(* IEC 61131-3 sources: ml2plc/benchmarks/st (part 21) *)

(* ---- ResNet2_straton.st ---- *)
FUNCTION_BLOCK ResNet2_FB

    (* Model Inputs/Outputs *)
VAR_INPUT
    input_data : REAL;
END_VAR

VAR_OUTPUT
    output_data : ARRAY[0..2] OF REAL;
END_VAR

VAR
    CONSTANT weights_0 : ARRAY[0..31] OF REAL := [0.446109116, -0.253379464, -0.341707826, 0.579259038, -0.196502939, 0.384631842, 0.528063476, -0.174200714, 0.4646855, 0.173207715, 0.330620855, -0.331686378, -0.31313917, -0.175854653, 0.48702389, 0.211235866, -0.0733348131, -0.239896551, 0.256497949, 0.395332277, -0.227466539, 0.452796817, -0.260912657, 0.231070071, -0.198892906, -0.148901105, 0.498160481, 0.427462339, 0.327300549, 0.239787996, -0.318450183, 0.391796708];
    CONSTANT bias_0 : ARRAY[0..31] OF REAL := [0.0780105293, 0, 0, -0.0437059142, 0, -0.0844902843, -0.0905284137, 0, -0.0596597679, 0.15236482, 0.109405488, 0, 0, 0, 0.0613273531, 0.0716272369, 0, 0, -0.0532285497, -0.055359453, 0, -0.0825184509, 0, -0.0527263731, 0, 0, -0.108202934, -0.0454206392, -0.0738661438, -0.0547046475, 0, -0.0875417367];
    CONSTANT weights_1 : ARRAY[0..1023] OF REAL := [-0.0672997385, 0.123918496, 0.0261855032, -0.207488403, 0.295382023, -0.205328912, -0.220387012, 0.309004188, -0.151001543, 0.397226214, 0.266850084, -0.0449176431, -0.0748620778, -0.0714222938, 0.0556719527, -0.21978052, -0.141455054, 0.0768866539, 0.148485273, 0.179841518, -0.120705262, 0.242057636, -0.0162528157, 0.0534217693, 0.107853472, 0.139660329, -0.0586810037, -0.0446375608, -0.244673312, 0.135248959, -0.0232865997, 0.291286677, 0.133107841, -0.0169415176, 0.072581023, -0.0316966772, -0.246254802, 0.156484276, 0.230665118, -0.022424221, 0.0690721869, 0.0099068284, 0.280228585, 0.282496542, 0.0474284887, -0.0939033031, -0.157858804, -0.0393083394, -0.200870991, 0.196391314, -0.0571665317, 0.0700698793, 0.0415192544, 0.283202559, 0.108373076, 0.18269524, -0.117297322, -0.287417442, -0.045781225, -0.200513572, -0.0697987527, 0.0264480114, 0.169026285, -0.0959516168, -0.0716886669, 0.297260195, -0.136756331, -0.189135864, -0.0970409364, -0.303627491, -0.0101010799, -0.273864031, -0.111413628, -0.124916166, 0.199581772, -0.264739096, 0.0937647521, -0.0471192598, 0.0671662092, -0.184105843, 0.2014893, -0.205362201, 0.273994476, -0.00908637047, -0.0441014767, -0.200558037, -0.0472564399, -0.0810055733, -0.137171343, -0.175276652, -0.303469598, 0.0569872558, -0.122404516, 0.132641941, -0.117922872, -0.0366746485, -0.271390259, -0.181193858, 0.154695168, 0.123995334, 0.300765067, -0.0419366695, 0.30564639, 0.0560056716, -0.13017562, 0.371984065, 0.0800307393, -0.243357852, 0.242418826, 0.2982063, 0.390265286, -0.29279983, 0.229600817, -0.105995312, 0.147868991, -0.282524794, 0.0784076452, 0.33515355, -0.0324381292, -0.127563611, -0.0404234231, 0.117910236, -0.268573463, 0.437732875, 0.205221027, -0.0789395124, 0.142241478, 0.318100512, -0.00765234232, 0.155244231, 0.229942471, 0.139751703, 0.167155415, -0.224905014, -0.253680557, 0.111216456, 0.166616023, 0.195199996, 0.26445052, -0.0218468606, 0.165077895, -0.305733055, 0.161665052, -0.280608475, 0.0925857723, -0.0801890641, 0.0903935134, -0.0246531367, 0.207986385, 0.244579464, -0.218942255, 0.254853576, -0.184336007, -0.259816915, 0.0658665895, 0.0739070773, 0.0859895349, 0.2244443, 0.303090066, -0.168849394, -0.117300168, -0.203983143, -0.516042411, -0.240961015, 0.320624799, 0.22011438, 0.155475706, 0.167489037, -0.223099396, 0.514761925, -0.0340227485, -0.135615855, 0.2276887, 0.100083739, -0.046878662, 0.00446370244, -0.16629912, 0.0464164019, -0.124795854, -0.211745948, -0.339682132, 0.560887516, -0.0539340675, -0.495146632, -0.154791906, 0.391963482, 0.0478856824, 0.300241709, -0.00436666375, -0.272856534, 0.473389745, 0.0918120444, -0.186532736, 0.169220388, -0.33542341, -0.13656354, 0.184764907, 0.121988617, -0.0807672292, 0.17290619, -0.0137443729, 0.403550833, -0.169839054, -0.199931324, 0.0710707009, 0.208184093, 0.194795758, 0.102081329, -0.135433197, -0.0341715217, -0.174149469, -0.269304931, -0.428490847, 0.436180294, -0.21050106, 0.136596486, 0.203933746, 0.305774748, 0.0526449233, 0.366092116, 0.38880232, -0.124543056, 0.399355233, -0.0542085133, -0.0242547095, 0.259555787, 0.169075102, -0.0785467029, -0.257587254, 0.0482283533, -0.303375334, 0.262526006, 0.195120007, 0.159601986, 0.0649527013, 0.289143413, 0.0153873265, -0.289190114, 0.184705019, 0.0448786616, -0.0187006891, 0.129755288, -0.000189214945, -0.12248905, -0.238008529, -5.98728657e-05, -0.159052655, -0.128630728, -0.127178386, -0.0828053951, 0.117196888, 0.291492611, 0.125405937, 0.0925316215, 0.24035868, 0.189899445, 0.0789665282, -0.114477828, 0.101446815, 0.0898142457, -0.0724863037, 0.267957658, -0.0225918293, -0.103431433, -0.176787034, 0.33514151, -0.276106536, -0.216690555, -0.0109675825, -0.237743527, 0.345496029, 0.0550661683, -0.281188637, -0.281930357, 0.0209647622, 0.173377007, -0.275085509, 0.442110121, -0.27953425, -0.269451231, -0.159710318, -0.0268889349, 0.261009961, 0.292426825, 0.00604014285, -0.039501071, 0.44544968, 0.385405064, -0.103716165, 0.197616503, 0.140080914, -0.190431833, -0.142311439, 0.338202953, -0.302250057, 0.00575613463, 0.237771541, 0.321618259, -0.248187274, 0.254863501, -0.0786112323, -0.256906897, 0.165188715, 0.00759845972, 0.196345091, 0.0205950439, 0.0259478632, 0.278409153, 0.269123256, -0.0704165474, -0.102515385, 0.143988624, -0.253235906, 0.00062259991, 0.0771465674, 0.102807239, -0.180491194, -0.0101891756, 0.108349077, 0.0780294985, -0.128736287, -0.236025348, -0.0358681642, -0.00330647826, -0.0861312822, 0.181077912, 0.117443472, 0.356189668, 0.188092053, 0.0508594029, -0.273949802, -0.00910276547, -0.274905294, -0.250903606, 0.241061077, 0.215696722, -0.0816203058, -0.21879968, 0.408205211, -0.246976987, -0.136179954, 0.320423037, 0.119813651, 0.349625587, -0.225764737, 0.353475153, -0.0903084055, -0.0600670241, -0.0816910192, -0.246967867, -0.125283241, 0.104817316, 0.194935232, -0.22541666, 0.139627814, -0.162285402, -0.139945656, -0.273778468, 0.154627442, -0.0709560364, -0.0483515859, 0.139850885, 0.26585874, 0.170851052, 0.0655213594, 0.275238186, 0.110014439, 0.241464347, 0.139358073, 0.225116462, 0.0450653136, 0.0663165748, 0.0984885991, -0.161821276, -0.253443301, -0.0401959717, -0.0450824797, -0.0893658102, -0.191750675, -0.114205316, -0.113555402, -0.032099843, -0.251139253, 0.0875837803, -0.0385817885, 0.14630121, -0.126950979, 0.15461868, 0.0945681036, 0.257601351, -0.131864205, -0.28712675, 0.231681079, 0.230294853, 0.261832148, 0.193466842, -0.301149845, -0.201477766, -0.236950368, 0.146894932, 0.042988807, -0.112412274, -0.255944818, 0.210005194, -0.0656734258, -0.126614377, 0.040821135, -0.045797646, -0.244730994, 0.25871709, -0.10164924, 0.0108816624, -0.263333112, -0.15512611, -0.265041053, -0.0407094359, 0.288093776, 0.244367093, 0.108738452, 0.0884629488, 0.125704706, 0.0346384346, 0.0489260256, -0.117135048, -0.0452102125, 0.123711288, 0.0750169158, 0.03458938, 0.0375772119, -0.160466671, 0.153726101, 0.299916059, 0.205223113, 0.099450469, 0.168587625, -0.170589864, 0.0105227232, -0.00761330128, -0.192904949, -0.0217333436, -0.0766484588, -0.236247391, 0.273411483, -0.171270818, 0.0562030673, 0.0808565915, -0.302630812, -0.171502382, -0.250153184, -0.201328039, 0.0215679221, -0.11872448, 0.342555076, -0.0201337449, -0.260737449, 0.308816582, 0.0652882904, 0.391782105, -0.11709775, -0.221956342, -0.125762343, -0.19962348, 0.0793167502, -0.301425576, -0.173867315, -0.0441781282, 0.120754406, 0.144720495, 0.0815581903, -0.196122408, -0.0626295954, -0.113548383, 0.175504923, 0.145190552, 0.0946770385, 0.151647747, 0.217094958, -0.203452721, -0.038656652, 0.101846643, -0.10814628, 0.108325951, 0.0775899515, -0.195024371, -0.241803467, -0.0457298718, 0.133528113, 0.42471084, -0.146245062, 0.120418303, -0.263231128, -0.14939186, -0.00569485081, -0.211991802, -0.110631473, -0.122159302, 0.211433142, -0.0213046074, 0.239424616, -0.172884226, 0.302616417, -0.0958690196, -0.198209673, 0.235887215, 0.201637536, 0.257626355, -0.261320055, -0.050790146, 0.1605165, -0.277989268, 0.27792275, 0.015366096, -0.21359621, -0.169574067, 0.255636603, -0.159326404, -0.242564619, -0.0658581853, 0.23809275, -0.0649103522, 0.0572633445, -0.233979613, -0.0433489978, 0.209428161, 0.100888282, 0.0781544745, 0.227146178, -0.216204301, 0.0940120816, -0.0834899247, -0.0717138499, 0.10444814, 0.0668695271, -0.227245539, -0.0815511048, -0.0642618835, 0.160572588, -0.186493456, -0.0400582254, 0.170362264, 0.274944872, -0.138044864, -0.0465166271, -0.0316170156, 0.141667455, -0.0781259239, 0.222043961, -0.292664409, -0.09773013, -0.267205209, -0.013055563, -0.268664062, -0.258037746, -0.233674765, -0.197328925, -0.181961954, 0.210466653, -0.074807182, 0.0213672519, 0.135242075, 0.29159227, 0.0965499282, -0.208291113, 0.170358896, -0.271036923, -0.0950112939, 0.118789613, -0.160189778, 0.0534884632, 0.165033877, -0.235269174, 0.0221406221, -0.0631530881, 0.175863415, -0.224407643, 0.23844102, -0.225643396, -0.149267823, 0.046709083, -0.22471258, 0.342396617, 0.382626325, 0.086022675, -0.111780778, 0.0649216473, 0.117322743, -0.22994262, -0.162323654, -0.309645176, 0.0411821902, 0.0823624283, 0.25201419, -0.16624178, 0.0215016305, -0.05505725, -0.279398203, -0.231971473, 0.473751515, -0.0695412159, 0.169299603, -0.216064066, 0.215218201, -0.102295764, 0.0126560032, 0.330998242, -0.238440096, -0.0759054124, 0.235605121, 0.0308294296, -0.205652803, -0.153373122, 0.21992442, -0.107053734, 0.449966788, -0.246368393, 0.303302258, -0.164613053, 0.281154096, 0.251495153, -0.0526953936, 0.128691703, -0.0415357351, -0.123309121, -0.125063479, -0.243296653, -0.200463638, 0.263173014, 0.0401532613, -0.0997288153, -0.00675202301, 0.272087842, -0.0488012917, -0.241687015, 0.2161116, 0.181204066, 0.383062124, -0.152072236, -0.175835103, 0.382474452, -0.0213172268, 0.0795238912, 0.293702573, 0.117500931, 0.302794188, -0.048030436, -0.0943690389, 0.280748278, 0.106655836, 0.27533105, -0.0209568441, 0.091119647, -0.0680115521, -0.0532403588, 0.00992289186, -0.135216832, 0.184090495, -0.198157549, 0.246385604, -0.183580667, 0.212307185, 0.134317905, -0.0904083997, -0.208351851, -0.00371128321, 0.016589433, 0.232418746, 0.173685908, -0.290628523, 0.275564283, -0.165179148, 0.177294314, 0.159701705, -0.0396937132, 0.0288962126, 0.0287567955, -0.0214288533, 0.406184524, 0.188659236, -0.137733087, 0.288018227, -0.376283169, 0.211254671, 0.0125238299, -0.182050586, -0.136293024, 0.244678944, 0.0101755811, -0.0860448629, -0.192576677, 0.144176096, 0.246334776, -0.0542725213, -0.319506258, 0.249152645, 0.300927252, -0.216155916, -0.263445467, 0.501632154, -0.0983170569, 0.490621924, 0.377952546, 0.182914823, 0.517102718, 0.292947888, 0.176778853, -0.0453032255, -0.292213202, 0.116734773, 0.0421213508, 0.0886447132, 0.164180636, 0.177889407, -0.0874125361, -0.28499952, -0.253518581, -0.0666396618, -0.191444427, 0.00308844447, -0.124373332, 0.0720646083, -0.201085448, 0.0728932619, -0.0851670355, 0.268443495, 0.291759223, -0.296979994, 0.15201956, 0.18446368, 0.128499776, 0.301611513, 0.200069577, 0.305754751, 0.23328355, 0.0512740016, 0.211027056, -0.0285782218, 0.28756842, -0.235887274, -0.201257139, -0.0654639155, -0.0219288748, 0.517582595, 0.142651647, -0.0918668807, -0.480128437, 0.445097446, -0.039173007, 0.206185371, -0.291620851, 0.289303392, -0.0353964828, -0.0932732373, 0.243763298, -0.168045878, 0.301816911, -0.454546899, -0.350679219, 0.389303118, -0.154629558, 0.0356258824, 0.217119068, 0.375954688, -0.216656104, 0.0966599658, 0.472218037, 0.24505803, 0.474726588, 0.287663907, -0.00348621607, 0.0777794719, 0.248905092, 0.304142505, 0.069024086, -0.00871711969, -0.17508626, 0.138942629, 0.0450723171, 0.222106844, 0.166393012, -0.285030186, -0.146981001, -0.173450544, 0.169468075, 0.101617634, 0.14248687, -0.211429179, -0.281644136, -0.21104835, 0.0707558692, -0.161577746, -0.179358691, -0.292363435, -0.0184406638, -0.0107237101, -0.0946408212, 0.119637281, 0.232440859, -0.188967675, -0.288388342, -0.0585837662, -0.0083989203, -0.189461887, 0.260625094, 0.0797997415, -0.0345056653, -0.273636639, -0.295552671, 0.111130029, 0.2143493, 0.0990378559, 0.0820131898, 0.219696254, -0.176936746, 0.194112211, -0.185160339, 0.20026961, 0.299959809, 0.132246137, -0.226150692, -0.165659562, 0.0304536223, 0.0551926792, -0.18758285, -0.00389325619, 0.120256096, -0.0793661326, 0.182034016, -0.0968718678, 0.210053414, 0.0536976159, -0.058866784, 0.032423377, -0.245521799, -0.0334720314, -0.476026595, 0.0220496655, 0.0105779376, 0.360177249, 0.226633102, 0.0757015273, -0.438258886, 0.176172927, 0.234365493, -0.22066617, -0.0561640561, -0.19579117, 0.355135053, -0.0497905016, 0.265808195, 0.0921390355, -0.219965175, -0.145613924, -0.043286223, 0.386870444, 0.10977602, -0.286260992, -0.0710007846, 0.302653104, 0.0277191214, 0.354971856, 0.129811853, 0.066929847, 0.00035183024, 0.216759875, -0.00531771779, 0.0594547167, -0.344661593, 0.29841271, 0.25737071, 0.322826356, -0.0608721077, 0.436551511, 0.163451761, -0.0346164703, 0.0586311519, 0.15674755, -0.115996219, -0.274861425, 0.0137932487, -0.306024313, -0.0696883276, -0.209392697, 0.0805150419, 0.0509290658, -0.110743746, 0.117124185, -0.110970736, 0.0164447147, -0.281959713, 0.179450154, 0.0630740449, -0.140035346, 0.324055582, -0.0899775475, 0.239219546, 0.400147587, -0.245016277, -0.0488338172, -0.457950622, -0.0780736506, 0.17666854, 0.395307273, 0.230418056, 0.454527378, -0.443111569, 0.103358082, 0.297938734, -0.270894229, 0.082223542, -0.0515313447, 0.152576774, 0.115509778, 0.130205333, -0.00376668572, 0.107549623, 0.0414021388, -0.118665934, 0.193046421, -0.00821468234, -0.455872506, -0.0179270804, 0.283343107, 0.0154615017, 0.157088995, 0.450618804, 0.226627737, 0.52094692, 0.0691082925, 0.00625914335, -0.190991536, -0.192506939, -0.114632443, 0.270887166, 0.426719934, -0.0118926466, 0.026724346, -0.384286642, -0.0412942842, -0.111217633, 0.153527528, 0.222803086, -0.186998546, -0.0981789753, 0.031683743, -0.136033341, 0.196271867, -0.295513868, -0.422320575, -0.319054574, 0.253908068, -0.0470398366, -0.359538227, -0.262141675, 0.556122601, -0.0490951799, 0.422659874, 0.243652195, 0.0135763288, 0.204732895, 0.504005373, 0.0145732462, -0.151889265, 0.295809776, 0.0527801514, -0.29109928, -0.0319833457, 0.00571236014, -0.108667865, -0.243677378, -0.187169373, -0.033985436, 0.0185488462, 0.0218675137, 0.078579098, 0.148238659, 0.0607049465, -0.0328954756, 0.164118737, 0.103054196, 0.0620963275, 0.228370219, -0.245889515, 0.00231522322, 0.00149768591, 0.207119197, -0.0681625307, -0.263822019, -0.0741106719, 0.303110272, 0.0252650976, 0.0528681874, 0.288920611, -0.0862795711, -0.183671564, -0.415967107, 0.0277608335, -0.0389414392, 0.509281099, -0.0653216392, 0.08415059, -0.146404579, 0.027331626, 0.0637321174, 0.0652593672, 0.119661465, 0.0570983589, 0.490790248, 0.0708687305, 0.0192686319, -0.135138795, 0.0672079623, -0.0580277219, -0.241328657, 0.495732963, 0.038197875, -0.444418669, -0.260325283, 0.0363532118, -0.0319354162, 0.21500051, 0.259890407, -0.136209637, 0.280829757, 0.164074123];
    CONSTANT bias_1 : ARRAY[0..31] OF REAL := [0, -0.00853045937, 0.126876727, 0, -0.0861710161, -0.0860414207, 0, 0.0468492433, 0.136715055, 0.0599241219, 0, -0.0130215548, -0.0051236595, 0, 0.0153312925, 0, -0.0135006029, 0, 0.184726223, 0.136625856, 0.102708332, -0.0912417546, 0, 0.150348634, 0, -0.0932127312, -0.00915876683, -0.0861517116, -0.0181769449, 0, -0.0608111285, -0.0683147013];
    CONSTANT weights_2 : ARRAY[0..1023] OF REAL := [-0.204679489, -0.135256469, 0.28196618, -0.0638390034, -0.174786299, 0.126281202, -0.209497452, 0.222915739, -0.0468465388, -0.216639012, -0.250750899, -0.280927479, -0.259657174, 0.0156140029, -0.235811859, 0.278314084, 0.0742395222, 0.290134758, -0.258248925, 0.0707915723, -0.302265584, -0.0793548822, 0.109813094, -0.20324108, 0.223869294, -0.052572906, 0.205616981, 0.102512896, -0.0969290286, 0.140410602, 0.241890162, 0.0239737928, -0.291626126, -0.216462642, 0.157533735, 0.21785447, -0.1888697, 0.0757077038, 0.222794265, -0.106055737, -0.192728728, -0.188463166, -0.182898849, -0.0930845514, -0.0597978532, 0.0867448747, -0.0387444645, -0.290577084, 0.0780397058, 0.0745291114, -0.172289535, 0.0823122859, -0.134248555, 0.252856761, -0.205714047, -0.102416694, -0.178794965, 0.0999448672, -0.00859764218, 0.243844897, 0.236200243, -0.113696873, -0.201874301, -0.113263831, -0.0378434174, -0.227657393, 0.0797862336, 0.333367527, -0.299939692, -0.0166706592, -0.125392675, 0.253749698, -0.355483234, 0.426590443, 0.558343112, 0.409482211, 0.187631369, 0.227338403, 0.285558254, 0.252233982, -0.349539638, -0.098085463, -0.0745894611, -0.260414094, 0.113806494, -0.36481443, -0.241131589, 0.0945619047, 0.452752471, 0.101931356, -0.30287379, 0.0321633108, 0.130271345, -0.0806449354, -0.210663259, -0.220049694, -0.17137076, -0.191594154, 0.301324457, -0.2250586, -0.253617704, 0.232058376, 0.077934593, 0.180609912, -0.139309749, -0.0280079544, 0.253463835, 0.244393975, 0.237231284, -0.20984596, 0.212327093, 0.264635891, 0.180089056, 0.218266934, 0.212391943, 0.280880839, 0.180849433, 0.106197894, 0.147727877, 0.018728435, 0.257006079, -0.206631452, -0.212920159, 0.166844428, -0.246302903, -0.00446945429, 0.247142047, -0.00678348541, -0.236221522, 0.277348638, 0.0965815783, -0.226228476, -0.0891875252, 0.40643695, 0.465085387, -0.152245566, 0.196031243, 0.140979126, -0.171359077, -0.0893353596, 0.454827428, 0.261000603, -0.299895495, -0.23500298, 0.0234229378, -0.060218025, 0.203745693, 0.122152202, -0.211209461, 0.0520563908, 0.10854879, 0.0593966246, -0.275008678, 0.0641941652, 0.481133044, -0.256873101, -0.285603046, 0.479949445, -0.135300189, 0.478868186, -0.406574875, 0.403340727, 0.0558100753, 0.225551426, 0.41712141, 0.00127660832, -0.0283386484, 0.0520305708, 0.500523508, -0.206790835, -0.362006932, -0.000284219335, 0.11284703, 0.130605608, -0.264846265, 0.133523747, 0.398929954, -0.00425994396, 0.44960174, 0.376377463, 0.2425109, 0.241941929, 0.246711314, 0.170248806, -0.264131367, 0.369570494, 0.443199039, 0.12817663, -0.182199731, 0.224466771, 0.257635802, 0.184784427, -0.0534651875, 0.114040047, -0.26297009, -0.137307927, 0.191011965, -0.224709436, 0.193394721, 0.134513915, 0.179350376, -0.188209772, 0.0368874371, -0.000262796879, -0.189553499, 0.11833626, 0.199825972, -0.168204218, 0.146432757, 0.232580811, 0.149660856, 0.122925818, 0.217384726, -0.143141761, 0.278794497, -0.0659557879, 0.2359505, 0.0733537376, -0.181416214, -0.24697648, 0.156488746, 0.163566709, 0.154782563, 0.16413027, -0.0641885176, 0.162349254, -0.165244937, -0.00756666251, -0.0619688965, 0.125170499, -0.164782301, 0.0368066728, 0.438915193, 0.369288772, -0.17342855, 0.372006238, 0.180813387, -0.0500442386, 0.181848824, 0.35768488, 0.33091262, 0.201537341, 0.0606543608, 0.183581203, -0.329741299, 0.19205898, -0.124992542, -0.203194737, 0.0749375671, 0.129340827, 0.0689797103, 0.0523179248, -0.232102171, 0.106971428, -0.164516747, -0.028096538, 0.26692003, -0.416765064, 0.146759704, 0.123076126, -0.313440531, -0.270631313, -0.449947, -0.0287845936, -0.411788732, 0.478075385, 0.478816599, 0.373561949, 0.0675536245, -0.204258502, 0.171388388, 0.416653246, -0.222486272, 0.212794915, -0.0879907608, -0.0584020466, 0.141890928, 0.153230354, -0.432367802, 0.197440714, 0.350558281, 0.383365989, -0.0781740323, 0.186996579, -0.195837736, -0.393867284, -0.12553376, 0.146623254, 0.07671763, 0.391239494, 0.192586288, 0.0520732291, 0.0479876958, -0.180293262, 0.0687054694, -0.309032947, -0.118887261, 0.162971631, 0.232025594, -0.115431778, 0.0105950609, -0.149042457, 0.275376558, 0.276807368, 0.161677882, -0.246772081, -0.0466549844, -0.0590618029, -0.0781350955, 0.0737073869, 0.299358219, -0.288225114, 0.166770518, 0.396302283, 0.349194467, -0.121977806, -0.203997999, 0.382262409, -0.154711246, 0.298326313, 0.0719448328, -0.0823758692, -0.230296239, 0.0475671887, 0.0851532519, 0.0975213349, 0.238155454, 0.174278498, -0.175005093, -0.265223473, -0.263997346, -0.198879018, 0.0115664899, 0.0591326654, -0.149858981, -0.109177634, -0.178252071, -0.00203052163, 0.268845469, 0.0775773823, 0.0275386274, -0.206349224, -0.136653408, -0.15385583, -0.155029312, -0.282329679, -0.222141564, 0.0748182833, 0.255190402, 0.171676189, 0.146660447, -0.149523973, -0.0342544094, 0.0865873992, 0.196472615, 0.0615327805, -0.201127067, -0.0292131901, 0.0689860284, 0.217757076, 0.220056325, 0.0298993532, -0.246281326, 0.0094137406, -0.205014378, 0.133170396, -0.00583136268, 0.230486065, -0.18984434, -0.265659779, 0.177857876, 0.21923694, 0.050457865, 0.178938717, 0.267668396, 0.179177284, 0.168444872, -0.172058687, -0.269957036, 0.198731601, 0.0808540285, -0.210361779, -0.203446448, -0.0371791422, -0.115300179, -0.0115000643, -0.15966849, -0.0855638981, -0.0802038908, 0.0730054528, 0.182234421, 0.0919757187, -0.0438024141, -0.284938186, -0.161267102, 0.0511448085, 0.201944143, 0.151732385, 0.11750789, 0.0223256852, 0.208975583, -0.0789252073, -0.249366164, 0.0771737546, -0.210034892, 0.0630125329, 0.282773703, -0.168602288, -0.228485093, -0.197542459, 0.227408201, 0.00968745165, 0.114427835, 0.251161247, -0.189475894, 0.0572520047, -0.0855299979, -0.012209028, 0.255862862, 0.0658447444, 0.279396147, 0.229320735, -0.0213460028, 0.0183748901, 0.0143043697, 0.175676167, 0.00535911322, -0.227714136, 0.210220248, -0.193221331, -0.244543672, -0.148611754, -0.190139264, 0.197188467, 0.112814814, 0.271459013, -0.28341198, 0.283254832, 0.194213003, 0.270252079, 0.0488406122, -0.137301132, 0.214347333, 0.213200539, -0.180703938, -0.128120601, -0.206830531, 0.0404673219, -0.0389949307, 0.0506746434, -0.0645795316, 0.0863745436, -0.00896019023, -0.200361013, -0.0323581994, 0.0325997397, -0.0739912689, 0.17362231, 0.0897462815, -0.12044479, 0.31924805, -0.27516371, 0.31264019, -0.11941921, 0.353853881, -0.0860883221, 0.218072325, -0.0713869631, 0.0661892593, 0.123493522, 0.154916063, -0.141882941, 0.142999113, 0.401889205, 0.386382669, 0.239116251, -0.228276312, 0.0787872225, -0.29939267, 0.00509946654, -0.115147322, -0.259926319, -0.0525318086, 0.0664702356, 0.0423623323, 0.1990951, 0.0846948028, 0.30295524, 0.181253284, -0.0447692871, -0.0963983834, -0.239262372, -0.053407073, 0.271961659, 0.0432170928, 0.129507035, -0.0613849461, -0.161630079, 0.223844141, -0.168244153, 0.131808519, -0.132705614, -0.0131464303, -0.0498532057, 0.0134880841, 0.205623835, 0.0286743045, -0.304037899, 0.297517449, 0.0676321685, 0.0823118389, -0.130943239, -0.0981799364, 0.0825493038, 0.092310302, 0.132190675, -0.0180039704, 0.222785085, 0.137986481, 0.289361268, 0.0720570758, 0.129101664, -0.140128732, -0.168845177, -0.126143813, -0.0213747621, 0.038553644, -0.303022981, 0.163347989, -0.20824483, -0.0491371453, 0.0485385358, -0.253569454, 0.0288275182, -0.0582758486, 0.0342372358, 0.00962677598, 0.231157124, -0.240408048, -0.21099937, -0.0426646173, 0.294546098, -0.245215863, -0.18224594, -0.0182284415, 0.135243684, 0.0727446079, 0.217568904, 0.166266769, 0.138461411, -0.2175951, 0.129577965, -0.230868846, -0.152226597, -0.131347224, 0.0510773361, 0.00408044457, 0.169953823, -0.0437824726, 0.163264632, -0.270352781, 0.212604791, -0.205052525, -0.202281937, -0.173584491, 0.248010248, 0.00338539481, 0.141827911, -0.117097601, 0.289717048, -0.261541098, 0.175698817, 0.103879333, -0.116942108, 0.125927597, -0.27946943, 0.133731633, 0.0409375429, 0.11390619, -0.0837004408, 0.199883446, 0.202443495, 0.146647006, 0.265037954, 0.18095395, 0.323377252, 0.111219957, 0.210307673, 0.0840765238, 0.301873416, 0.252628654, 0.176735342, -0.225448921, -0.00881180167, 0.264034539, -0.0576801077, -0.207668871, -0.0362603888, 0.183284, -0.222751856, 0.029674856, 0.253859907, -0.301360816, 0.276103348, 0.159531534, 0.09506578, 0.296914607, -0.0876111984, -0.218210489, -0.224868655, -0.276840299, 0.170778424, -0.0902170613, 0.026544407, 0.0524329469, 0.139356345, 0.337209821, 0.343271613, 0.106872618, 0.247088611, -0.146878138, -0.140349343, 0.319549531, 0.265812397, -0.0614267886, 0.176764369, -0.295758694, 0.00160560687, 0.142407343, -0.17890656, 0.00188067136, -0.179448411, 0.323931873, 0.14950569, 0.112876579, -0.0789793506, -0.254204988, -0.249873608, -0.111487955, 0.233570397, -0.0383268632, -0.220227048, 0.188659593, 0.138276428, -0.391264945, -0.219422072, 0.119032457, -0.324904621, -0.149002716, 0.260387927, 0.512180686, 0.343798786, 0.246067539, -0.213445902, 0.343288749, -0.0358869024, -0.0598138869, 0.0849777758, -0.229632109, 0.0804907382, -0.207954884, -0.246657565, -0.152553603, 0.230183572, 0.258402884, 0.605133116, -0.000907221751, 0.40813598, 0.138139337, -0.394745469, -0.245143875, -0.356614888, -0.278564036, 0.51167649, -0.167552158, 0.0385506786, 0.30153054, 0.178012431, 0.491966486, -0.226964116, 0.249466941, -0.31189698, -0.212363005, 0.12730749, 0.107616968, 0.245273083, -0.0632424355, -0.107013598, 0.400151312, -0.126116946, 0.443775713, 0.0567636304, -0.0484892353, 0.225377142, 0.17650643, -0.16261822, -0.350496858, 0.21365118, 0.0242102928, -0.272912949, 0.144263998, 0.183707282, 0.235746235, 0.106295653, -0.0331136882, 0.117457211, -0.0399730206, 0.0439910293, 0.0704419613, -0.169385076, 0.137371719, 0.183431178, 0.0584154129, -0.266066253, 0.0112705529, -0.0212856233, 0.223700017, -0.0228022039, 0.0189183056, -0.0324111879, -0.155158073, -0.22306934, 0.11734134, 0.288133234, 0.275658756, -0.179903343, 0.296819836, -0.187510654, -0.154961348, 0.275978237, 0.267136604, 0.1356273, 0.0229957998, -0.166162252, -0.0112787187, 0.271157116, 0.504267514, -0.0745441094, -0.128601953, 0.396112651, -0.0514549389, -0.0184277389, -0.0510308333, -0.151744619, 0.0578206517, 0.451091677, 0.449969262, 0.439691722, -0.121170506, -0.107776523, 0.201376095, 0.392380595, -0.37306577, -0.182681888, -0.082582891, -0.0752992257, -0.0241405126, 0.154176563, 0.0456010364, -0.200354218, 0.186367407, 0.0181775708, -0.202771991, 0.154682621, -0.182058185, -0.219726712, 0.059972316, -0.343565434, 0.209741443, -0.222851798, -0.199444413, -0.02868554, 0.235248834, -0.304307938, 0.161286384, 0.201732069, -0.0422318876, -0.157119676, -0.224580228, 0.067997545, -0.125626177, 0.0241714716, -0.0759897828, -0.0502993762, -0.296199769, 0.243887156, -0.267505169, 0.138399065, -0.233483225, 0.246404737, -0.174308226, -0.137947485, 0.101638436, 0.124087334, -0.114575863, 0.096797049, 0.0372642577, 0.0244682431, -0.10504967, 0.0597021282, -0.243710384, 0.346117526, -0.191104233, 0.00756108714, 0.360030293, 0.254576176, 0.380814731, -0.170184657, 0.0216305014, 0.169229582, -0.0979294181, -0.174209282, 0.345129073, 0.113265961, -0.108804695, 0.363609046, 0.212997556, -0.033747524, -0.068172805, 0.198910668, 0.258692235, 0.252833068, 0.2392544, -0.0721322894, -0.333581597, 0.0375342928, -0.110548787, 0.326079488, 0.0975811481, 0.314479381, 0.147384316, 0.424212158, 0.162820056, 0.279910028, -0.149647564, -0.113421351, 0.122204378, 0.0914485157, -0.11268647, 0.0712843239, -0.0754816532, -0.113101743, 0.129354239, -0.0762300938, -0.294329286, 0.018773675, 0.0962105021, -0.0627630502, -0.139184624, -0.0883929282, 0.192166761, -0.0048656296, 0.0775612146, 0.014094159, -0.227728426, 0.16301775, 0.248803243, 0.139576599, -0.236111104, -0.134085178, -0.0108638359, 0.0713160485, 0.000784546137, 0.0634449497, -0.285768718, 0.540881157, -0.0152861401, 0.196317405, 0.0716606081, -0.118341036, 0.377459377, 0.0323503166, 0.503604591, -0.325088292, -0.351278603, -0.345217735, 0.345662981, -0.115596712, -0.213419259, -0.0567794181, 0.110530913, -0.281917006, 0.269924909, 0.134860232, -0.183613077, 0.222686723, 0.22196804, 0.130703807, -0.137397841, 0.095159784, 0.382972747, -0.257635623, -0.114726156, 0.219153389, -0.274423659, 0.193779275, -0.378756016, 0.55745393, -0.273371994, 0.153506696, 0.347348154, -0.0390162319, -0.0190924518, 0.0466835201, 0.338260919, -0.289644122, -0.045777481, -0.0979495496, -0.109888777, -0.159528181, -0.315120131, 0.0249667857, 0.3593283, -0.266355038, 0.329570562, 0.0659172311, 0.141647443, 0.172656283, 0.413104653, -0.0921770632, -0.309635311, 0.0745841414, -0.0158826876, 0.159715265, 0.280772299, 0.185895413, -0.224144131, 0.0355212055, -0.0401628911, 0.258820683, 0.020608902, -0.00089943409, -0.126454577, -0.187050238, 0.0248265862, 0.21769926, -0.039658457, -0.193980694, 0.191328883, 0.251601726, 0.238136321, 0.247954696, -0.122940779, 0.133804053, 0.12044853, -0.00639125705, 0.084846288, -0.250858724, 0.184372365, -0.0337354839, 0.173017561, 0.185794771, -0.136319786, -0.154326752, 0.161565125, -0.0733977556, -0.261118054, 0.237281889, -0.284483045, 0.259607047, -0.118910857, 0.319470137, -0.0940027982, 0.167246327, 0.15437226, 0.423810035, 0.453898102, 0.2123539, 0.515671432, -0.263677806, -0.384399831, -0.276800603, 0.440641314, -0.115233019, 0.273297697, -0.149060681, 0.187632188, -0.0750807822, 0.393690765, -0.15505597, -0.0574740916, 0.110269904, 0.451854825, 0.121877313, -0.311037689, 0.205216989, -0.07337486, 0.234148517, -0.108864084, 0.344401598, -0.256927043, 0.349292517, 0.078679502, 0.375678301, 0.0557315461, -0.0197441522, 0.360949874, 0.00126973551, -0.0796471536, 0.139007911, 0.465253472, -0.00500912592, -0.220044911, 0.330124229, 0.211857736, -0.23185648, 0.00514952559, 0.0121980738, 0.425808966, 0.210433066, -0.138632327, 0.10696023, 0.0690508857, 0.253821135, -0.0823103711, 0.180217087, -0.0521651581, -0.0492838956, 0.231640503, -0.0903923362, -0.19418329, 0.404094219, 0.151551336, 0.41822511];
    CONSTANT bias_3 : ARRAY[0..31] OF REAL := [0.15151085, -0.00549688889, -0.0278635602, 0.164689794, -0.0236758217, -0.00926770084, -0.0640082359, -0.0109293507, 0.0096361218, 0.18045342, 0.167336062, 0.183991253, 0.00347143412, 0, 0.145016342, 0.156027064, -0.0661333054, -0.00646232022, -0.0596447811, -0.0291018039, -0.0106637869, -0.0447131656, -0.0726215765, 0, 0.0979361758, 0.220422715, -0.0577485524, 0.053236004, -0.0165364016, -0.0795688108, 0, -0.0443540327];
    CONSTANT weights_6 : ARRAY[0..1023] OF REAL := [0.0423009433, -0.125790134, 0.226051986, -0.0357659571, 0.216817826, -0.358196169, 0.113928027, -0.296048373, 0.354682565, 0.104639202, 0.0836121291, 0.38464427, 0.09730196, 0.0722192526, -0.107720353, -0.188351095, -0.297569394, -0.0126603991, 0.279470056, -0.187208816, 0.173353896, -0.0451729298, 0.240580156, -0.383692145, 0.428899467, -0.25482446, 0.134113222, 0.518396139, -0.305747777, 0.165480375, -0.13187553, -0.0798858255, -0.0843793899, -0.0530831814, -0.349667042, -0.202598363, -0.0539790243, 0.42323938, 0.296966612, -0.225120366, 0.0834762231, 0.434091777, 0.19163458, -0.267244548, 0.42511943, -0.10342706, -0.257457256, 0.221439674, -0.211297899, -0.0577185526, -0.110783815, 0.0277600363, 0.253185958, 0.0685807467, 0.132226005, 0.0041287099, 0.325069249, 0.257862478, 0.167387515, -0.325158834, 0.384652436, -0.332001626, 0.365253597, -0.194888949, -0.180765018, 0.275981158, -0.0959078521, 0.241078928, -0.169195786, 0.0800399408, 0.170336306, -0.265964568, -0.249380469, 0.251532733, -0.203793287, -0.182373986, -0.283105522, 0.182440251, 0.31397751, -0.00957679749, 0.075581938, 0.28843084, -0.0690082312, 0.118075877, 0.168982834, -0.0824798197, 0.101467103, 0.203187943, 0.17364642, 0.0646778718, -0.00096732378, 0.0401217528, -0.026663661, -0.227451354, 0.089766793, 0.299514562, -0.329149902, 0.0847316682, 0.238331869, 0.152660891, -0.102428906, -0.209868148, -0.0361074507, -0.264742672, 0.24686192, 0.195887923, -0.0490344577, 0.339129806, 0.321493864, 0.154694334, 0.139662385, -0.0378654823, 0.0556175858, -0.180449381, -0.257891923, 0.241288692, -0.0935784653, -0.1163297, 0.00155670941, 0.337323457, 0.183867663, 0.132523268, 0.299205154, -0.0655880645, -0.0818198547, 0.28338024, 0.212773114, 0.0941432416, -0.570614398, -0.288114667, -0.0787712783, -0.234560788, 0.291475266, 0.388435811, -0.184467867, 0.0161492527, -0.124954529, -0.0790996775, -0.288120806, -0.251139522, -0.0881813616, -0.0902432874, -0.0650542527, 0.316850722, -0.0104520731, -0.254874259, -0.244556203, -0.24943167, 0.162652522, -0.0661111325, -0.209356561, 0.0419312939, 0.146880999, 0.0992746502, 0.143128425, -0.18333517, 0.357891113, -0.328243315, 0.279128373, -0.0311047137, -0.201804623, -0.233284876, -0.0154908476, -0.13330698, -0.265543371, 0.411796123, 0.199394181, -0.0530769825, -0.394122511, -0.0533640347, -0.436150432, -0.136589125, 0.447410434, -0.349607825, -0.767117381, 0.361389458, 0.0190853905, 0.168821484, -0.286791474, 0.191248387, -0.0722396076, 0.20492819, -0.168038502, -0.0610720478, -0.0322836637, 0.229064777, 0.276264817, -0.188246489, -0.0029287287, -0.281597942, 0.485978961, -0.089131251, -0.454895794, 0.0885980725, -0.583386481, 0.249597982, 0.093602933, 0.401051074, 0.182700485, 0.111778408, -0.426135391, 0.404733658, -0.319206327, -0.135104164, 0.16884166, -0.269442499, -0.677988231, 0.0933919996, -0.110211551, 0.0533670858, 0.274164677, -0.034223672, -0.0645384192, 0.251852781, 0.0273246858, 0.496946633, 0.0339165628, 0.108153924, -0.135926679, -0.219843075, 0.210196838, 0.144822106, 0.307614803, -0.0304114819, 0.134284928, 0.0461441278, 0.0190904066, 0.0106084915, 0.0963880122, -0.138905436, -0.178883806, 0.0350694358, -0.161462411, -0.226585031, -0.168459147, 0.217511848, 0.00232085912, -0.192238122, -0.185177505, 0.278003603, 0.165126503, 0.0706270933, 0.0398160443, -0.0480608046, -0.0824743807, -0.21219781, -0.21391806, -0.305020243, 0.191144735, 0.292650759, 0.206448823, 0.0859370977, 0.0968351886, 0.0571502261, 0.156657591, 0.0889105797, 0.0787278637, -0.125621796, -0.048659727, 0.132065356, 0.241339967, 0.0302367527, -0.200879022, -0.168844506, -0.0636498183, 0.391604245, 0.176699132, -0.0634741113, 0.349128932, -0.164361373, -0.442244589, 0.337881058, 0.194366217, 0.0232700482, 0.0419569351, -0.1305013, -0.0122175394, 0.0366523862, -0.0360458605, -0.101712011, 0.268878162, 0.358265698, -0.28440544, 0.0753252208, 0.226901263, 0.0454228148, 0.0869102031, -0.0431394875, 0.138498962, 0.0179591477, 0.0707068667, 0.0545778498, -0.227329016, 0.161272004, 0.219899163, 0.266284436, 0.170998976, 0.0461607575, 0.550597429, 0.387942731, -0.257321209, 0.420359045, 0.335143536, -0.0522419401, -0.143776849, -0.292115062, 0.24676089, -0.186925456, -0.0909894556, -0.12318109, -0.304902047, 0.222862214, 0.177171841, -0.0675419271, -0.00998198241, 0.157330796, 0.151477307, 0.287911505, -0.0747540295, 0.106006265, -0.0908687264, -0.227996647, 0.00245764968, 0.24865739, -0.113826834, -0.389270723, -0.341020525, 0.104753941, 0.261327326, -0.197135881, 0.511418104, 0.284275919, -0.0961943343, 0.455836266, 0.100646339, 0.243058845, -0.247537196, 0.197578713, -0.246891603, -0.279520124, 0.0799680874, -0.150676951, 0.207488194, -0.142935142, 0.133621603, -0.0261798259, -0.212552786, 0.258970141, -0.387301117, 0.268923998, -0.162345812, -0.248713821, 0.166159257, -0.234904915, -0.0506722964, 0.136956081, -0.0161326919, 0.237550795, -0.158257529, -0.270248592, 0.00648764102, -0.0811474323, 0.271124631, 0.23387076, 0.0228706282, 0.428895444, 0.234345809, -0.193682402, -0.277639538, -0.0542408489, -0.184264317, -0.0607525595, 0.0243354775, -0.0618640482, -0.0741198882, 0.0695161149, 0.409474939, -0.102613024, -0.299581379, -0.0302265771, -0.0905358568, 0.224896714, -0.0254502371, -0.0784858167, -0.0960717201, 0.242310971, -0.133200958, -0.187372297, -0.284839481, 0.0373332985, 0.0939624384, -0.16979906, 0.134718105, 0.0443862602, 0.144108161, 0.219357878, -0.0544792525, 0.126239464, -0.336690068, 0.143944621, 0.0834249109, 0.127459735, 0.179903641, 0.125341117, -0.195693061, -0.0123710334, 0.223720968, 0.279200464, 0.309253842, 0.0955327377, -0.166285902, -0.214190856, -0.150016502, -0.0221532062, 0.176856473, 0.0403885543, 0.10900864, 0.0844879746, -0.0256391466, 0.190568119, -0.0756136775, -0.168081284, 0.228286117, 0.184770495, 0.0794119835, 0.101312399, 0.0174291432, -0.229970217, -0.107041851, -0.0299378633, -0.147796124, 0.135027617, -0.076323539, 0.196455389, -0.136140868, -0.15242961, -0.297595322, 0.268853277, -0.306081772, -0.235011339, 0.0682312846, 0.0281739533, -0.262217879, -0.0421818793, 0.24620387, 0.00353482366, 0.0282435119, 0.143977046, 0.119495705, -0.304054767, 0.214439899, -0.0573004, -0.0426736698, -0.00534119923, 0.232765377, -0.298282832, 0.463601798, 0.12735717, 0.128070861, -0.0716682747, -0.048194468, 0.449055582, -0.132900998, 0.00517642405, 0.124559343, -0.0519258119, -0.156628609, -0.278578043, -0.0213215817, -0.27828303, 0.0387053452, 0.0462420285, 0.377790481, 0.175675839, -0.263917774, 0.209180012, -0.19289954, -0.223212153, 0.106517792, 0.163594157, -0.221901819, -0.188828021, -0.0661086887, -0.190387979, -0.0855609626, -0.0792594999, -0.0224655531, -0.191546261, 0.390218973, -0.182257563, 0.0761514753, 0.267081141, -0.0730520561, 0.195442915, 0.1261985, 0.324406445, -0.236988112, 0.0551995896, 0.0264911, 0.228242666, -0.180638194, -0.162573323, -0.252948046, -0.163001031, 0.344733059, 0.195890233, 0.178869903, 0.154100791, 0.10623233, -0.120936655, 0.0172378756, -0.152924851, -0.454507291, -0.228110462, -0.333555669, -0.241648883, 0.261162728, 0.343055844, 0.35510847, 0.140914083, -0.395139039, 0.493091226, -0.103029147, -0.0748043135, 0.424542844, -0.454302132, -0.416242003, 0.445887506, 0.217544511, -0.0344426595, 0.131312326, -0.192004547, -0.176152796, -0.221430913, 0.171940222, 0.266956776, 0.381788284, -0.0122210849, 0.0751685426, -0.318172663, 0.441737533, 0.156246081, 0.104305185, -0.293639868, -0.221548617, -0.249040216, -0.235861868, 0.277391106, 0.0219161212, 0.0634618551, 0.0392980725, -0.0183740854, -0.0568681881, 0.00934559107, -0.142207995, -0.0807104632, -0.20466511, 0.0248596147, -0.16451551, 0.149044007, 0.17448312, -0.0527889132, -0.211640745, 0.252037615, -0.107537679, 0.203633457, -0.0208883584, 0.302550614, -0.00199513696, 0.0422494709, 0.123262793, -0.182073951, -0.0718897134, 0.274784088, 0.185307637, 0.016862452, -0.402763665, -0.0663023293, -0.479049653, 0.21997948, -0.19869785, 0.485822797, 0.325658202, -0.168805525, -0.495869309, 0.261673659, -0.221560389, -0.428493202, 0.379379392, -0.469475716, -0.48414737, 0.0475211814, 0.25103724, 0.246232197, 0.169537723, 0.195288733, -0.285054207, -0.230555326, -0.0827380866, 0.234976038, 0.532914817, 0.295589656, -0.212547272, 0.162255287, 0.419421703, -0.175461367, 0.21505025, 0.185273707, -0.335693091, 0.147099704, -0.462255776, -0.255811274, 0.224329144, -0.0124325594, 0.205371261, 0.0318574011, -0.109709941, 0.0107474187, -0.288051963, -0.0442421474, 0.0988274366, -0.36958921, -0.513040721, 0.333079785, -0.0538684875, -0.270858347, -0.187043905, 0.0551031269, 0.056669414, -0.00255042315, 0.118919633, 0.229129359, 0.260899723, -0.0010361243, 0.27428931, -0.15735206, -0.00179547234, 0.0291315299, 0.0568751395, -0.0997283012, -0.190779671, -0.218523234, -0.112121858, 0.322309703, 0.206250161, -0.107823908, -0.0462691225, 0.0836636722, -0.197753936, -0.276076794, -0.207480028, -0.282821298, -0.0265177134, -0.247018337, -0.0979018733, -0.243366033, 0.299129993, 0.102958031, -0.221814767, 0.0849224925, 0.154980227, -0.106702983, -0.169575453, -0.155088782, -0.261757523, -0.273117304, 0.106121846, 0.297675759, 0.289185077, 0.155774966, -0.0959317684, 0.0692664385, -0.223100066, -0.122799665, -0.327967435, -0.317192882, 0.0993198901, 0.282140434, -0.0140098343, 0.131905884, -0.347699583, 0.392752528, 0.220863894, -0.273349524, 0.349267483, -0.0185028333, -0.479156345, 0.334563673, 0.0530006774, 0.268007904, -0.299093872, -0.174457282, 0.0596756935, -0.0261847675, 0.256202579, 0.340914726, 0.271126807, 0.459985256, -0.170322567, -0.0740677267, -0.0700618699, 0.110616066, 0.349578977, 0.12270996, -0.28840366, -0.223576546, -0.376913935, -0.00889683142, 0.174228996, 0.288166434, -0.0926035792, 0.0564029515, -0.312326223, -0.108814351, -0.336783767, -0.422059119, 0.147130847, -0.112820074, -0.462775379, 0.286943793, -0.225329861, 0.199072585, 0.0262849331, 0.0572461337, 0.0196778774, 0.0365224481, -0.298687965, 0.2957955, 0.0718266293, 0.248218864, 0.165144593, 0.208500594, 0.350200236, -0.339656055, 0.112521388, -0.0694022924, -0.30071184, -0.0400292277, -0.26554051, -0.273952723, -0.085234046, 0.24783203, 0.265917629, -0.240497112, -0.275556624, 0.243338794, -0.197343603, -0.293294489, 0.241594642, 0.294589788, -0.270102978, -0.0805493891, -0.141567439, 0.260685593, -0.0584824383, 0.0103724301, 0.241969794, -0.219980463, 0.139372885, 0.201815456, -0.129380301, -0.109165221, -0.247791752, -0.166421473, -0.254870683, 0.229641408, -0.14008297, 0.082115829, 0.216543972, 0.243624538, -0.115283772, 0.128091365, -0.0125387684, -0.112591699, -0.303687096, -0.239466846, 0.192435205, -0.264854044, 0.366258979, 0.333079666, 0.0547362603, 0.712514818, 0.420474559, -0.442672163, -0.278284639, 0.235130087, -0.156521425, 0.00912833214, 0.136461109, 0.183566451, 0.223094463, -0.18576695, -0.287605226, -0.378859192, -0.154404134, 0.226181909, -0.252294451, 0.471755594, -0.225533873, 0.0991383195, 0.188798636, 0.235263199, 0.0377827771, 0.108561836, 0.0202547144, 0.236043692, -0.0238635391, -0.184035391, 0.27792713, -0.114163101, -0.00627177488, 0.095444411, 0.0818532407, 0.358962864, 0.00885722879, -0.117014825, 0.292946726, 0.152037829, -0.0793638676, 0.27496171, -0.00204696273, 0.0733370781, 0.211719334, 0.203182101, 0.401544392, 0.129787788, -0.0615753792, 0.344649017, 0.396610051, 0.232138321, 0.00247897534, -0.232831538, -0.274918139, 0.0712967217, -0.140307426, -0.155776829, -0.312981665, 0.451258421, -0.0611403547, -0.0937829912, -0.348439723, 0.256666154, 0.00332944212, -0.36961621, 0.468926221, 0.0165066961, -0.36621663, 0.50422132, -0.192109123, 0.220578969, -0.0636099502, -0.0225161277, -0.0138186216, 0.162092894, 0.0845716596, -0.0670932084, 0.221348569, 0.207287028, -0.258025855, -0.268616766, 0.0833133236, 0.0906072631, -0.0970331952, -0.302971363, 0.227304041, 0.0701878369, 0.103975438, -0.321448207, -0.284966111, 0.0546144396, 0.202484027, 0.192938596, 0.405504107, -0.120458379, -0.0995231941, 0.0176873077, -0.114662506, 0.299742699, 0.106414162, -0.163575932, 0.0854470432, -0.111256771, -0.22295922, -0.0171526223, -0.101826482, 0.0775648355, -0.168530032, 0.191495821, 0.490707844, 0.347011179, 0.263281316, -0.0198134352, 0.38279748, 0.284762532, 0.217713609, -0.0966390669, 0.274289995, -0.294971675, -0.131608486, -0.0882483497, 0.110222839, -0.302902013, 0.133009627, 0.09202075, 0.0521754324, 0.22471115, 0.113432527, 0.0434851572, 0.242308497, 0.10426081, -0.00738954544, 0.113250218, 0.0809162855, -0.0213614851, 0.252549976, -0.248513728, 0.235877782, -0.0581952631, 0.26298061, -0.0510342345, -0.108697504, -0.169658944, -0.265481323, -0.119629472, -0.168868601, 0.147454306, -0.234578624, 0.148263484, -0.418611586, -0.300675213, -0.00871061161, 0.128228858, 0.247511044, 0.345100015, 0.22982879, 0.0828597248, -0.0861068368, 0.461450547, -0.243431032, -0.304843843, 0.45811829, -0.260032356, -0.286119521, 0.25225845, -0.273061275, -0.121072449, -0.0245819669, 0.125408977, -0.212921172, -0.203906059, -0.205443576, 0.491495579, 0.218547136, 0.442893356, 0.0343887247, -0.275091708, 0.291343957, 0.102542974, 0.0203316752, -0.00634527206, -0.244422123, -0.249972135, -0.261188954, 0.0179378986, 0.221036226, -0.253236353, -0.18469736, -0.227377743, 0.302024156, 0.0104332268, 0.0571029484, 0.284029514, 0.0533148944, 0.00642812252, -0.00143432617, -0.0420979261, -0.0503995419, -0.114822313, 0.255191594, -0.216471195, 0.242331654, 0.0167051256, -0.226628989, -0.19661054, -0.264778316, -0.1843777, 0.25669679, 0.172157854, 0.127889901, 0.269744009, -0.203344822, -0.174746886, -0.305384725, 0.256571501, -0.415793508, 0.0293531418, -0.307875067, -0.04958345, 0.00131417031, -0.269373626, -0.207887754, 0.130413279, -0.00960878842, 0.0802605823, 0.373825133, -0.0580155328, -0.472687095, 0.485479474, 0.194238052, -0.182139128, -0.053170111, -0.171621591, 0.0708632469, 0.0144039392, -0.261881024, 0.298481733, 0.0884690955, 0.449684829, 0.0680728704, -0.143362433, 0.456231087, -0.020072611, 0.320502847, 0.0488895178];
    CONSTANT bias_6 : ARRAY[0..31] OF REAL := [0.046065066, 0, -0.0190256666, -0.0534179136, -0.00336124306, -0.00999941025, -0.0601420403, 0, 0.177893505, 0.035768088, 0.229685664, 0.179855481, -0.0841028988, 0.175335124, 0.0450567603, 0.014103503, -0.00015270352, -0.0198834073, -0.0095967995, -0.00921531487, -0.0128452741, 0, -0.0109253274, -0.0661542937, 0.146812245, -0.0134299155, -0.00511262612, 0.173508465, -0.0358441025, 0.0460290201, -0.0524213314, 0];
    CONSTANT weights_7 : ARRAY[0..1023] OF REAL := [0.696965337, -0.425572038, -0.0124750175, -0.454262227, 0.00770199299, 0.673409045, -0.35552901, 0.133035973, -0.405757964, 0.435457647, 0.176012516, -0.259070784, 0.0526116639, -0.179251224, -0.685974419, -0.557297349, 0.026896745, 0.083768189, 0.06145823, -0.0420161486, -0.0770936161, -0.517920494, 0.302174181, -0.109914497, 0.454531014, -0.401484787, 0.196335629, 0.114402629, 0.484787554, -0.419739991, 0.131457701, -0.525040388, 0.0218699276, -0.00843754411, 0.130763501, 0.0453180373, -0.261570454, 0.231266171, 0.14041248, -0.150360554, 0.21441862, -0.106453612, 0.301262468, 0.128003359, -0.269974202, 0.00775644183, 0.118737757, -0.200946987, -0.144442409, -0.270234376, -0.236532301, -0.268752098, -0.0458901525, -0.290161818, -0.0426600277, -0.293334991, -0.143675834, 0.123336792, 0.223108441, -0.0152406096, -0.167314708, 0.0709961951, -0.112513095, -0.0946361572, 0.352671236, 0.0633277148, -0.100119464, -0.328425974, -0.03042835, 0.264760464, -0.100179784, 0.252682835, -0.118299723, 0.379216075, 0.158170924, -0.245778188, 0.237490535, 0.36283347, -0.136392534, -0.399134129, 0.0126428902, -0.0975233912, 0.0260714591, 0.109776437, 0.022193227, 0.110348985, 0.618779898, -0.301410973, 0.000802389113, -0.1210026, -0.269414127, 0.146038741, 0.155972809, -0.0195733532, 0.11079029, -0.149775863, -0.0188240875, -0.130381867, 0.234488532, 0.00693501998, 0.13113755, -0.125127271, -0.224939346, 0.192458794, -0.251354158, -0.0559266582, 0.115683667, -0.131063834, 0.186389178, 0.0575638562, 0.0515241176, -0.177111626, -0.213718995, -0.260617942, -0.311560392, -0.121136598, -0.136864081, 0.158393279, -0.247277722, -0.213672429, 0.319099247, 0.0424774252, -0.217664108, 0.0733582303, 0.0865076482, 0.189959049, -0.113231719, -0.167562768, 0.121859923, -0.107053503, 0.21689482, -0.306519896, -0.139735192, -0.0525539219, 0.137694538, 0.277069569, -0.0124758091, 0.0584755465, 0.00664382521, 0.176539853, -0.248395681, 0.273150414, 0.212669566, 0.297428697, 0.22037378, -0.134781465, 0.00648336159, -0.301100731, -0.226388007, 0.280572951, 0.107294366, -0.142516777, 0.0114334822, 0.177158341, -0.259080857, -0.186600402, 0.143441409, -0.138016999, -0.210677966, -0.183829799, 0.0103514018, 0.322654486, 0.434209317, -0.211887494, -0.0989680812, -0.709826529, -0.0314815529, 0.316612095, 0.0355967321, 0.0909824297, -0.0161110815, 0.141115546, 0.411118567, 0.491116852, 0.0815100297, 0.158555105, 0.00380989909, 0.0325110443, -0.0139920739, 0.173851699, -0.0830620155, 0.510648847, -0.341825187, -0.00457854243, -0.635425448, 0.278676569, 0.443823487, 0.312433481, -0.250826329, 0.0924364626, -0.252370417, 0.27807641, 0.00292166462, 0.17300576, 0.175417289, 0.188273698, -0.256306589, -0.231017292, 0.311479211, 0.101328477, -0.087451756, -0.253629625, -0.215819553, -0.382644147, -0.106965065, 0.257888138, -0.0935752764, -0.0360229649, 0.0615254641, -0.25007984, -0.0403431132, -0.190366521, 0.0989143848, 0.183037266, -0.00106490438, -0.195043325, 0.000767204154, 0.471863508, -0.0329909995, 0.034967944, -0.240443826, 0.330452263, -0.183411777, -0.0518309809, 0.0119438171, 0.243542343, 0.281483442, -0.268857062, -0.0288396478, -0.0803266019, -0.299922556, 0.0745203495, 0.00863289833, -0.119709402, -0.273133069, -0.237470582, -0.116267875, -0.0103208125, 0.0487196445, -0.0837379098, 0.077483505, 0.252253979, 0.0389327705, -0.0804390162, -0.287603378, -0.154697731, -0.23082009, -0.0285177231, 0.0736643374, 0.181847066, -0.0232335031, -0.184853941, 0.106023729, -0.0366936922, -0.290526092, 0.0300653875, 0.167654172, -0.274094939, -0.366497815, 0.502952218, -0.0707105771, 0.232042566, -0.328350991, -0.455214351, 0.193826467, 0.426049173, 0.266488731, 0.519607842, -0.203651413, -0.204463676, 0.304759532, 0.341860801, 0.0368262529, -0.220895708, 0.0676381811, -0.246637106, 0.179857954, 0.0694600418, 0.479727328, -0.168309957, 0.411688477, -0.295417756, -0.340031832, -0.0663810447, 0.344733894, 0.032624092, 0.166009933, -0.308683455, -0.431732535, 0.480302334, 0.391812414, -0.0258753747, -0.155325428, -0.69197309, 0.143985361, 0.159691051, 0.0586706549, -0.0478923395, 0.182829171, 0.114467956, 0.0696068555, 0.459607065, 0.0855634958, 0.236511499, -0.155534834, 0.194287702, 0.309163451, -0.297604054, -0.365406543, 0.10110756, 0.0814178362, -0.149148315, -0.207489669, 0.284899205, 0.0963382497, 0.142904967, -0.110910818, 0.383015066, -0.102222472, -0.00579420384, 0.443447202, 0.116973169, -0.568473756, 0.430070162, 0.0534169972, -0.15302898, -0.569367051, -0.060554821, 0.138348266, 0.581483901, 0.532705963, 0.0795565397, -0.105224222, 0.038537547, 0.387009233, -0.163335249, -0.102199659, 0.0823252574, -0.371436357, 0.00202056766, 0.147038251, 0.0980918705, 0.296901047, 0.249531776, 0.30156821, -0.00228712521, -0.408944219, -0.0487018228, 0.121689036, 0.0753933713, 0.175764695, 0.108644582, -0.0149587188, 0.10152211, -0.314113587, -0.194645077, -0.235040978, 0.0125054736, -0.343776405, -0.555387557, -0.386055857, 0.467185915, 0.355092227, 0.762303412, -0.827248633, 0.0659005567, -0.00991847552, 0.168695077, 0.0125243366, -0.214904383, -0.658762932, -0.257405967, 0.579136789, -0.234206975, 0.455616534, 0.0611006245, 0.339377671, -0.480572373, -0.911797643, -0.390998006, 0.401130319, -0.381678641, -0.347490251, -0.105943128, -0.28553462, 0.0159271341, 0.240740597, 0.00333705219, 0.0582735315, -0.686321437, 0.383500308, 0.413927883, -0.0309322532, -0.183925778, -0.353048503, 0.120974191, 0.320696801, 0.41828379, -0.113802485, 0.0911439732, -0.125538424, 0.162278593, 0.328606784, -0.0427318439, 0.04242111, 0.295007288, 0.0182766002, 0.117341086, -0.656848967, 0.111713633, 0.326780766, -0.176031604, -0.249191374, 0.285160422, 0.029264899, 0.403999984, 0.423614979, 0.172128424, -0.347453147, 0.0410611369, 0.0250360053, 0.310506284, -0.600645542, -0.189122587, 0.162287816, 0.232688621, 0.208908603, 0.250347167, -0.111579634, -0.301809251, 0.473928899, 0.407907754, -0.00877436996, -0.0534283519, -0.457796752, -0.216536999, 0.36930716, 0.0234591272, 0.330734104, -0.140827909, 0.178206548, -0.0701909587, -0.415120661, -0.587533772, 0.400556803, -0.293752581, 0.156959668, -0.35017845, 0.509965599, -0.580648124, -0.154729292, -0.52914232, -0.113128483, 0.334058642, 0.117303051, 0.0228555296, -0.515133619, 0.246055439, 0.319413483, 0.033750508, 0.0412687846, 0.193547741, -0.406977922, -0.36664027, -0.0483321548, 0.168110132, -0.290306151, 0.248343199, -0.31926617, -0.093695201, 0.457288653, -0.270948082, 0.327385664, -0.193126842, -0.277083963, -0.275356948, 0.636034131, -0.155900344, -0.185263753, -0.0742744729, -0.129384637, 0.60393399, 0.171084613, -0.143731296, 0.0920975655, -0.47300148, 0.386613846, -0.0452283844, 0.248413906, -0.0453487635, -0.130735949, 0.0689658523, 0.0691124722, 0.140205935, 0.169704899, 0.306278348, -0.2284545, -0.0786308572, -0.0898166895, -0.243578494, 0.00569618214, 0.444122344, -0.112142526, -0.259075701, -0.510384321, 0.189697579, 0.435087621, 0.308014095, -0.0443768725, 0.276326567, 0.157689556, 0.292997569, -0.209561259, 0.177630454, 0.266212583, -0.189523682, -0.141224623, -0.294096619, 0.186715022, -0.206432164, 0.28385064, -0.0970800668, -0.233691931, 0.204295799, -0.212764367, -0.169756532, 0.289480776, 0.10397166, -0.0893522352, -0.292596161, 0.100929961, -0.252269149, 0.0703386068, -0.00896264054, 0.116490453, -0.0523757339, 0.181890279, 0.22511971, 0.254319489, 0.178610951, -0.115120456, -0.123811118, 0.164738446, -0.251088381, -0.139749333, -0.206608936, -0.247167125, -0.243351653, 0.0491047502, 0.248196512, -0.0223228633, -0.137623042, -0.175845459, 0.064390853, 0.186741725, 0.0204023384, -0.150762156, -0.0579429679, 0.246738479, 0.224769995, 0.233293146, -0.161801592, -0.027525099, 0.152252898, 0.283100456, 0.0640011281, 0.0288589597, 0.0565277226, 0.246870786, -0.00058200187, 0.133958265, -0.0840905011, 0.00257615116, -0.0693306401, 0.019505484, -0.0362477414, 0.261339724, 0.0660063401, 0.158006608, -0.0845215321, -0.0950676501, 0.183873788, -0.210932925, -0.280518889, -0.2290418, -0.268612385, 0.0994316787, -0.199969187, 0.0599627569, -0.152291462, -0.198237866, -0.135641858, -0.0936126858, -0.186587125, -0.203803629, 0.285384685, -0.297869265, -0.14777711, 0.0950407088, 0.185630977, -0.294005573, -0.155923128, -0.0303075463, 0.0306556225, -0.207352132, 0.289859891, 0.00876015425, -0.035254769, -0.166374385, 0.224656418, 0.0365344882, 0.18270275, -0.193076134, 0.0523616374, 0.088819854, -0.257332146, -0.0887077674, 0.107509702, -0.211296469, 0.227283135, 0.187960997, -0.0550236255, 0.202599376, 0.148077354, -0.212565452, 0.232545376, -0.251226038, -0.292171538, -0.265042692, -0.222401917, 0.000110954046, -0.0648710504, 0.0769141018, 0.273979336, -0.240394369, -0.0309286248, 0.174879059, 0.126584247, -0.0568807423, 0.105581313, 0.0393341146, -0.252430141, -0.174195692, 0.203471616, -0.268663675, 0.173340723, 0.263071984, -0.134033203, -0.248103619, -0.217972159, 0.12414214, 0.0926405862, 0.150795326, -0.2161486, -0.2995359, 0.18589358, -0.121494129, 0.116116971, -0.27156204, -0.08181113, -0.0163346343, 0.21491766, -0.183056653, 0.161056817, 0.174699455, -0.0756241232, -0.300119519, -0.219501853, 0.0957794785, 0.0586510003, 0.129047051, 0.106559753, 0.251048893, -0.272713304, 0.181690335, 0.1188896, -0.0186873078, -0.201658949, -0.0394966304, 0.162966728, -0.00398737192, 0.00541430712, 0.286092132, 0.169025481, 0.0938329995, -0.0404688418, 0.197128624, -0.012212038, -0.0768416226, -0.227206409, -0.0605284274, 0.120017916, 0.242930681, -0.163972005, 0.0343070924, 0.0950588286, -0.283331245, 0.119762182, 0.265106887, -0.0367939174, -0.0890540928, -0.0754073113, -0.121581942, 0.0240540206, 0.165571913, -0.0788320303, 0.207621664, -0.0608751401, -0.236746848, -0.229722992, -0.309312493, -0.199644804, 0.246266425, -0.0388333313, -0.231182873, -0.28938666, -0.0852914229, 0.127132192, 0.219269186, -0.24605763, -0.010866195, -0.142100185, -0.266323447, 0.26336512, -0.263663352, -0.0106320577, 0.1183649, 0.0248650014, 0.0896441415, -0.0368609205, -0.221683547, 0.16726467, 0.185754329, -0.0466969982, 0.100290127, 0.258109629, -0.353465974, 0.126338392, -0.113909215, -0.188452274, -0.194115311, -0.17864804, 0.196741164, 0.0597201474, 0.206435919, -0.0926698819, 0.191386208, 0.118541375, 0.0108582275, 0.123223342, 0.0203074664, 0.184328318, -0.0781305879, -0.0412917919, -0.182512492, -0.186976776, -0.0690055043, 0.407485723, -0.153934166, 0.101274781, 0.0300630219, 0.213275805, -0.0704917535, 0.0985206589, -0.195325136, 0.385939896, 0.220668882, 0.441593409, 0.318906814, 0.516893208, 0.00302047026, 0.246910304, -0.0343478061, 0.211347491, -0.224081829, -0.075066492, 0.282728493, 0.0514900349, 0.323377848, 0.148849085, -0.0540174879, 0.270508736, 0.179961666, -0.0142629566, -0.272535712, 0.095599927, 0.10564328, -0.207949072, 0.311026305, 0.276351869, 0.144048631, -0.264415205, -0.182311937, 0.47848478, -0.00634554215, -0.278761476, -0.421602428, 0.486623317, -0.31333527, 0.314758718, -0.0402104147, 0.142329782, -0.181337923, 0.233083189, -0.218328774, -0.198587954, 0.151959121, -0.0403886698, 0.237960577, 0.000396092131, -0.386091083, -0.22716257, -0.202574566, 0.469723493, 0.22511667, -0.0485011414, -0.23309961, -0.145659015, -0.0504665487, 0.236505777, 0.03145919, 0.156357527, -0.324489534, 0.136566207, -0.418168277, 0.300612271, 0.308621079, 0.0192018449, -0.00402103737, 0.365092486, -0.314835578, 0.408390015, 0.00832532439, -0.00207912503, -0.199070662, 0.112644672, -0.274405181, 0.266614765, -0.12923871, 0.022493396, -0.0482205711, -0.253843725, 0.11145328, -0.158875361, 0.137883201, 0.193825305, -0.0869452953, -0.188784227, 0.196680158, -0.19173643, -0.185577244, -0.00177709165, 0.161155775, 0.0399096236, -0.152769983, 0.079197593, 0.0402290225, 0.0904241726, 0.00207823934, 0.0752336606, -0.19206135, 0.257340044, -0.214997351, 0.0654263273, 0.206675172, -0.346203685, -0.305421114, -0.138736844, -0.242514983, 0.401338905, -0.334246397, -0.536974669, 0.174231291, 0.313181788, 0.37326315, 0.777741671, -0.724793971, -0.196852624, -0.0113996528, 0.190205157, -0.101818815, -0.0731762052, -0.67447269, 0.304049045, 0.380955279, 0.00464151194, 0.505375028, -0.073581934, 0.0330387354, -0.267104745, -0.428916097, -0.465622813, -0.0341051184, 0.0174973067, 0.0592112727, 0.098631002, -0.0514589548, 0.263129473, 0.293475986, 0.316690475, -0.0897324234, -0.617124617, 0.240499303, 0.415535361, 0.451071352, -0.430378288, -0.30219692, -0.10279952, 0.241131514, 0.407398283, -0.182798669, 0.278176427, 0.2107943, -0.0544432625, 0.274078876, 0.171579182, 0.0168831125, 0.582827747, -0.267883271, 0.232941583, -0.198801219, 0.284586132, 0.202702582, 0.348091543, -0.253476113, 0.550308883, -0.270993322, 0.425108671, 0.338867635, -0.11253576, -0.206026614, 0.0577263832, -0.0562936515, 0.169156313, 0.160081729, -0.383194476, -0.196228907, 0.252097577, 0.240194216, 0.0299131051, -0.0534505285, -0.0208027642, -0.0221766979, 0.267329842, -0.290644437, -0.0993616134, -0.405614763, -0.233593687, 0.317183614, -0.258464456, 0.148786247, 0.0562397018, -0.188056841, -0.00285600196, 0.0271013733, 0.0560174584, 0.142336175, 0.154277325, 0.159117386, 0.322743207, -0.0304633845, 0.0810233429, 0.327721715, 0.260459393, 0.28296721, -0.429413438, 0.422827661, -0.0342015848, 0.403933138, -0.378505558, -0.339093983, -0.0479762331, -0.170190975, 0.400465161, -0.224378809, 0.00213353406, 0.264918298, -0.117029347, 0.177011371, 0.174274415, -0.0583742969, 0.155514762, 0.18779999, -0.159250617, -0.414283961, 0.579815805, -0.140579313, 0.171675146, -0.336225599, 0.153423682, -0.237003818, 0.0958352163, 0.143583268, -0.289194405, 0.298214346, 0.138118744, 0.032494843, 0.231931239, -0.0158346891, 0.0180291533, -0.131696448, 0.282267302, 0.1432769, 0.0832591653, -0.100443333, 0.298321813, -0.291152805, 0.108140498, -0.269369751, -0.0559225976, 0.276901871, 0.175810128, 0.0156878829, 0.0704467893, -0.295131922, -0.15239808, 0.105308324, -0.11231716, 0.124838561, -0.0991676599, 0.207252592, 0.254895777, -0.0838771164, -0.000925213099];
    CONSTANT bias_8 : ARRAY[0..31] OF REAL := [0.141434908, 0.0432733782, -0.124192744, 0.120511875, -0.000832263904, -0.0289485268, -0.137065947, -0.129716218, 0.0822892487, 0.167498499, 0.138521075, 0.154646561, -0.149244398, 0.0518487953, 0.129266709, 0.0929838195, 0, -0.0130553758, -0.0956565365, -0.0108651146, 0.170342505, -0.0352739841, 0.119917497, -0.0197882541, 0.0404277593, 0.00698901713, -0.150984779, -0.134503573, 0.0457827225, 0.0124715837, -0.0172215924, -0.0206808355];
    CONSTANT weights_11 : ARRAY[0..95] OF REAL := [0.498224497, 0.0502187572, -0.593330979, -0.522627413, 0.458213657, 0.249259174, 0.0720091537, -0.383112788, 0.548259437, -0.0533615239, 0.481050968, -0.0924307778, 0.124834575, -0.430146515, -0.11986199, 0.287840724, -0.799370825, 0.204687238, -0.22228162, -0.372063994, 0.301369935, 0.0614436641, -0.485295773, 0.462331802, -0.587614357, 0.180880338, -0.156508088, 0.315634191, 0.085335426, -0.605618, 0.414695352, -0.0716700181, -0.703150809, 0.204102322, 0.300819486, -0.478523195, 0.0813441947, -0.119165942, 0.638306379, -0.681795955, -0.178639486, 0.218786493, -0.124697737, 0.566166699, -0.509519637, 0.13568005, 0.533299565, 0.119743563, 0.336455554, -0.34957993, -0.411417395, 0.1551245, 0.366843879, -0.0861211196, 0.0359399468, -0.845785916, 0.136662394, 0.31982258, 0.112232365, -0.240569293, 0.393351048, 0.516565263, 0.0558515973, -0.46442309, 0.317726195, 0.25089094, 0.52674073, -0.0834692344, -0.711942554, 0.0820730627, 0.0769959465, -0.174524337, 0.672163546, -0.487948388, -3.02611206e-05, -0.459344417, 0.150462016, 0.261800498, -0.355333507, -0.578431726, 0.247226343, 0.145157427, -0.200589418, 0.560618281, 0.393166453, -0.0303138644, -0.0382165052, -0.34001863, 0.415801167, 0.490103513, -0.160248145, 0.222737715, -0.237386137, -0.721500874, -0.12006399, 0.279553384];
    CONSTANT bias_11 : ARRAY[0..2] OF REAL := [0.0486483872, 0.0960481763, -0.144294515];
END_VAR

VAR
    (* Merged variables from all regions *)
    buffer_0 : ARRAY[0..31] OF REAL;
    buffer_1 : ARRAY[0..31] OF REAL;
    buffer_2 : ARRAY[0..31] OF REAL;

    (* Temporary computation variables *)
    i : DINT;
    j : DINT;
    t : DINT;
    sum : REAL;
    (* Computation helpers *)
    max_val : REAL;
    exp_val : REAL;
    exp_sum : REAL;
    (* Spatial loop variables *)
    oc : DINT;
    oh : DINT;
    ow : DINT;
    ic : DINT;
    kh : DINT;
    kw : DINT;
    ih : DINT;
    iw : DINT;
END_VAR

(* Forward pass execution *)

(* Region: r0 [ACYCLIC] *)
(* Acyclic Region r0 *)
(* Layer 0: Fused Linear + RELU *)
FOR j := 0 TO 31 DO
    sum := 0.0;
    FOR i := 0 TO 0 DO
        sum := sum + input_data * weights_0[i * 32 + j];
    END_FOR;
buffer_0[j] := MAX(sum + bias_0[j], 0.0);
END_FOR;

(* Layer 1: Fused Linear + RELU *)
FOR j := 0 TO 31 DO
    sum := 0.0;
    FOR i := 0 TO 31 DO
        sum := sum + buffer_0[i] * weights_1[i * 32 + j];
    END_FOR;
buffer_2[j] := MAX(sum + bias_1[j], 0.0);
END_FOR;

(* Layer 2: MatMul *)
FOR j := 0 TO 31 DO
    sum := 0.0;
    FOR i := 0 TO 31 DO
        sum := sum + buffer_2[i] * weights_2[i * 32 + j];
    END_FOR;
buffer_1[j] := sum;
END_FOR;

(* Layer 3: Add (Bias) *)
FOR i := 0 TO 31 DO
    buffer_2[i] := buffer_1[i] + bias_3[i];
END_FOR;

(* Layer 4: Add (Element-wise) *)
FOR i := 0 TO 31 DO
    buffer_1[i] := buffer_2[i] + buffer_0[i];
END_FOR;

(* Layer 5: Activation (RELU) *)
FOR i := 0 TO 31 DO
    buffer_0[i] := MAX(buffer_1[i], 0.0);
END_FOR;

(* Layer 6: Fused Linear + RELU *)
FOR j := 0 TO 31 DO
    sum := 0.0;
    FOR i := 0 TO 31 DO
        sum := sum + buffer_0[i] * weights_6[i * 32 + j];
    END_FOR;
buffer_2[j] := MAX(sum + bias_6[j], 0.0);
END_FOR;

(* Layer 7: MatMul *)
FOR j := 0 TO 31 DO
    sum := 0.0;
    FOR i := 0 TO 31 DO
        sum := sum + buffer_2[i] * weights_7[i * 32 + j];
    END_FOR;
buffer_1[j] := sum;
END_FOR;

(* Layer 8: Add (Bias) *)
FOR i := 0 TO 31 DO
    buffer_2[i] := buffer_1[i] + bias_8[i];
END_FOR;

(* Layer 9: Add (Element-wise) *)
FOR i := 0 TO 31 DO
    buffer_1[i] := buffer_2[i] + buffer_0[i];
END_FOR;

(* Layer 10: Activation (RELU) *)
FOR i := 0 TO 31 DO
    buffer_0[i] := MAX(buffer_1[i], 0.0);
END_FOR;

(* Layer 11: Fused Linear + SOFTMAX *)
FOR j := 0 TO 2 DO
    sum := 0.0;
    FOR i := 0 TO 31 DO
        sum := sum + buffer_0[i] * weights_11[i * 3 + j];
    END_FOR;
output_data[j] := sum + bias_11[j];
END_FOR;

(* Softmax: find max *)
max_val := output_data[0];
FOR i := 1 TO 2 DO
    IF output_data[i] > max_val THEN
        max_val := output_data[i];
    END_IF;
END_FOR;

(* Softmax: compute exponentials and sum *)
exp_sum := 0.0;
FOR i := 0 TO 2 DO
    output_data[i] := EXP(output_data[i] - max_val);
    exp_sum := exp_sum + output_data[i];
END_FOR;

(* Softmax: normalize *)
FOR i := 0 TO 2 DO
    output_data[i] := output_data[i] / exp_sum;
END_FOR;

END_FUNCTION_BLOCK
